PROGRAM CallHardware
VAR
	i : DINT;
END_VAR

//conveyors
ForceSetLifterConveyors();

FOR i:=0 TO 20 BY 1 DO
	allConveyors[i]();
END_FOR

//robots
FOR i:=1 TO 6 BY 1 DO
	robots[i]();
END_FOR

//A23
wrapperA23();

//A22
cardboardSkidLeft();
cardboardSkidRight();
cornerGuardMagazineLeft();
cornerGuardMagazineRight();

insertionA22Left();
insertionA22Right();
insertionA22Bottom();
wrapperA22();

//A21
chipboardSkidLeft();
chipboardSkidRight();

woodBunkMagazineLeft();
woodBunkMagazineRight();

stagingTableLeft();
stagingTableRight();

strapperA21();

insertionA21Left();
insertionA21Right();
insertionA21Bottom();

(*
//paper
Hardware.wrapperPaper();

//cardboard + corner guard
FOR i:=Surface.LEFT TO Surface.RIGHT BY 1 DO
	Hardware.insertionCardboardCornerGuardSides[i]();
END_FOR
Hardware.wrapperCardboardCornerguard();

//wood bunk
FOR i:=Surface.LEFT TO Surface.RIGHT BY 1 DO
	Hardware.insertionWoodBunkSides[i]();
	Hardware.stagingTable[i]();
	Hardware.woodBunkMagazine[i]();
END_FOR

Hardware.strapper();
*)

END_PROGRAM

(* stored: Version 1.1.0.1, ProductVersion 3.1.4024.11
   POU CallHardware: Id {37cad5aa-fa76-4d83-b429-cad99db8cb21}, SpecialFunc None *)
